FUNCTION_BLOCK CheckComponentsEnabledVisitor IMPLEMENTS I_ComponentVisitor
VAR
	Enablable : I_Enablable;
	_Enabled  : BOOL;
END_VAR

METHOD Check
VAR_INPUT
	Components : I_ComponentCollection;
END_VAR
_Enabled := TRUE;
Components.Accept(THIS^);
END_METHOD

{attribute 'monitoring' := 'call'}
PROPERTY Enabled : BOOL
GET
Enabled := _Enabled;
END_GET
END_PROPERTY

METHOD VisitComponent
VAR_INPUT
	Component : I_Component;
END_VAR
IF __QUERYINTERFACE(Component, Enablable) THEN
	IF NOT Enablable.Enabled THEN
		_Enabled := FALSE;
	END_IF
END_IF
END_METHOD

END_FUNCTION_BLOCK

(* stored: Version 1.1.0.1, ProductVersion 3.1.4026.18
   POU CheckComponentsEnabledVisitor: Id {b6aa3a03-aef9-42fd-8c69-693977a88be7}, SpecialFunc None
   Method Check: Id {f77fa282-8b96-4dc7-afde-10508d1c86dd}
   Property Enabled: Id {6b77e7fa-dd4c-43e8-8659-ad40c4de7aab}
   Get Get: Id {563920ab-7755-43c0-afe9-f898f10fd9c0}
   Method VisitComponent: Id {70521ac0-123c-42b7-9b30-6a97e4735e8c} *)
